fbCamSwitchPulserSearch();
fbCamSwitchPulserSync();
fbInMotionTimer();
fbTestTimer();
fbMotionStage();

IF nTestStep = 78 THEN
    TEST_FINISHED();
ELSIF fbTestTimer.Q THEN
    AssertTrue(FALSE, CONCAT('Timed out at step: ', TO_STRING(nTestStep)));
    TEST_FINISHED();
END_IF
END_METHOD

END_FUNCTION_BLOCK

// ---- POUs/FBs/Common/FB_LimSwStatus.TcPOU
FUNCTION_BLOCK FB_LimSwStatus IMPLEMENTS I_LimSwStatus
VAR_INPUT
END_VAR
VAR_OUTPUT
END_VAR
VAR
    (* Hardware *)
   // NC Forward Limit Switch: TRUE if ok to move
    bLimitForwardEnable AT %I*: BOOL;
    // NC Backward Limit Switch: TRUE if ok to move
    bLimitBackwardEnable AT %I*: BOOL;
    // NO Home Switch: TRUE if at home
    bLimitHome AT %I*: BOOL;
END_VAR

PROPERTY LimitBackwardEnable : BOOL
GET
LimitBackwardEnable := bLimitBackwardEnable;
END_GET
SET
bLimitBackwardEnable := LimitBackwardEnable;
END_SET
END_PROPERTY

PROPERTY LimitForwardEnable : BOOL
GET
LimitForwardEnable := bLimitForwardEnable;
END_GET
SET
bLimitForwardEnable := LimitForwardEnable;
END_SET
END_PROPERTY

PROPERTY LimitHome : BOOL
GET
LimitHome := bLimitHome;
END_GET
SET
bLimitHome := LimitHome;
END_SET
END_PROPERTY

END_FUNCTION_BLOCK

// ---- POUs/FBs/DS402/FB_HomeDS402.TcPOU
FUNCTION_BLOCK FB_HomeDS402 IMPLEMENTS I_HomeDS402
VAR_INPUT
END_VAR
VAR_OUTPUT
END_VAR
VAR
    iMotionLogger : I_MotionLogger;
    //iLimSwStatus : I_LimSwStatus;
    //iHomeShareData : I_HomeShareData ;
    bCommandMoveHome  : BOOL;
    bBusy	: BOOL;
    bDone	: BOOL;
    bError 	: BOOL;
    bAbort   : BOOL;
    bAborted  : BOOL;
    nErrorID : UDINT;
    fOffset  : LREAL;
    fPosition	: LREAL;
    rtDone	: R_TRIG;
    fHomeSpeedFast	: LREAL;
    fHomeSpeedSlow	: LREAL;
    bBit13OpModeSpecific	: BOOL;
    bBit12OpModeSpecific	: BOOL;
    bTargetReached	: BOOL;
    nDriveControl : UINT := 15;
    nModeOfOperation : SINT;
    nModeOfOperationDisplay : SINT;
    nMostRecentModeOfOperation : SINT;
    eHomeMode: E_EpicsHomeCmd :=E_EpicsHomeCmd.AUTOZERO;
    rtExec: R_TRIG;
    ftExec: F_TRIG;
    bMove  : BOOL;
    tonSyncHoming : TON;
    {attribute 'hide'}
    eHomeState	: E_MoveState;
    rtReset: R_TRIG;
    bReset: BOOL;
    sMessage: T_MAXSTRING;
END_VAR

//NB: The calling must pass drive status register.
THIS^.rtExec(CLK:=THIS^.bCommandMoveHome);
THIS^.ftExec(CLK:=THIS^.bCommandMoveHome);
// an interruption can be external i.e, an halt, Reset or a local condition
THIS^.rtReset(CLK:=bReset);
tonSyncHoming(PT:=T#50MS);
CASE THIS^.eHomeMode OF
    E_EpicsHomeCmd.AUTOZERO:
        THIS^.bMove := TRUE;
    E_EpicsHomeCmd.NONE:
        THIS^.bMove := FALSE;
        THIS^.bBusy := THIS^.rtExec.Q;
        THIS^.bDone := NOT THIS^.rtExec.Q;
    ELSE
        THIS^.bMove := FALSE;
END_CASE

IF THIS^.bMove THEN
    IF THIS^.bBusy AND THIS^.ftExec.Q THEN
        THIS^.eHomeState := E_MoveState.ERROR;
        THIS^.bAborted := TRUE;
    END_IF
    CASE eHomeState OF
        // Wait for a rising edge
        E_MoveState.IDLING:
            IF THIS^.rtExec.Q THEN
                THIS^.bDone := FALSE;
                THIS^.bBusy := TRUE;
                THIS^.bError := FALSE;
                THIS^.nErrorID := 0;
                THIS^.bAborted := FALSE;
                THIS^.eHomeState := E_MoveState.INIT;
                // make sure the run flag is clear, this would be the case
                // in EnableMode ->ALWAYS and ModeofOperation ->CSP
                //nDriveControl:=15;
                THIS^.tonSyncHoming.IN := TRUE;
            END_IF
        E_MoveState.INIT:
            // sdo write homing paramters;
            // This mode will be restore after homing
            THIS^.nMostRecentModeOfOperation := nModeOfOperationDisplay;
            nDriveControl:=31;
            // take some time for drive to register above commad and start
            // homming routine.
            IF tonSyncHoming.Q THEN
              eHomeState:=E_MoveState.STARTED;
            END_IF

        E_MoveState.STARTED :
            // this is a comfirmation that routine is ongoing
            IF NOT bTargetReached
               AND NOT bBit13OpModeSpecific THEN
                bBusy:=TRUE;
                bDone:=FALSE;
                eHomeState:=E_MoveState.IN_PROGRESS;
            END_IF
        E_MoveState.IN_PROGRESS :
            // Genral Motion error i.e Following error ?
            IF bBit13OpModeSpecific THEN
                eHomeState:=E_MoveState.ERROR;
            // Reached
            ELSIF bTargetReached
                AND bBit12OpModeSpecific
                AND NOT bBit13OpModeSpecific THEN
                eHomeState:=E_MoveState.REACHED;
            END_IF

        E_MoveState.REACHED:
            bBusy:=FALSE;
            bDone:=TRUE;
            //prepare next move
            nDriveControl:=15;
            // Restore default mode
            //nModeOfOperation:=THIS^.nMostRecentModeOfOperation;
            tonSyncHoming.IN := FALSE;
            eHomeState:=E_MoveState.IDLING;
        E_MoveState.ERROR:
            bError:= TRUE;
            bDone:=FALSE;
            // sdo read in case of error
            bBusy:= FALSE;

    END_CASE
END_IF

IF THIS^.rtReset.Q THEN
    THIS^.bError := FALSE;
    THIS^.nErrorID := 0;
    THIS^.bAborted := FALSE;
    THIS^.sMessage := '';
    THIS^.bReset := FALSE;
    THIS^.eHomeState := E_MoveState.IDLING;
END_IF
//NB: The calling must forward control register for i/o update.
// Reset execute after when done successfull or after abort reset
// this way the done and error condition is latched till next move or global reset.
rtDone(CLK:=bDone);
IF  rtDone.Q  THEN
    THIS^.bCommandMoveHome := FALSE;
END_IF

PROPERTY Aborted : BOOL
GET
Aborted := bAborted;
END_GET
END_PROPERTY

{warning 'Add property implementation'}
PROPERTY Active : BOOL
GET
END_GET
END_PROPERTY

{warning 'add property implementation'}
PROPERTY Busy : BOOL
GET
Busy := THIS^.bBusy;
END_GET
END_PROPERTY

METHOD PUBLIC CallAfterInit
VAR_INPUT
    iMotionLogger : I_MotionLogger;
END_VAR
THIS^.iMotionLogger := iMotionLogger;
END_METHOD

{warning 'Add property implementation'}
PROPERTY CommandMoveHome : BOOL
SET
bCommandMoveHome := CommandMoveHome;
END_SET
END_PROPERTY

{warning 'add property implementation'}
PROPERTY Done : BOOL
GET
Done := THIS^.bDone;
END_GET
END_PROPERTY

PROPERTY DS402Control : UINT
GET
DS402Control := nDriveControl;
END_GET
END_PROPERTY

PROPERTY DS402ModeOfOperation : SINT
GET
DS402ModeOfOperation  := nModeOfOperation;
END_GET
END_PROPERTY

METHOD DS402Status
VAR_INPUT
    ModeOfOperationDisplay : SINT;
    Bit13OpModeSpecific	: BOOL;
    Bit12OpModeSpecific	: BOOL;
    TargetReached	: BOOL;
END_VAR
nModeOfOperationDisplay := ModeOfOperationDisplay;
bBit13OpModeSpecific := Bit13OpModeSpecific;
bBit12OpModeSpecific := Bit12OpModeSpecific;
bTargetReached := TargetReached;
END_METHOD

{warning 'add property implementation'}
PROPERTY Error : BOOL
GET
Error := THIS^.bError;
END_GET
END_PROPERTY

{warning 'add property implementation'}
PROPERTY ErrorID : UDINT
GET
ErrorID := THIS^.nErrorID;
END_GET
END_PROPERTY

//FB_Init is always available implicitly and it is used primarily for initialization.
//The return value is not evaluated. For a specific influence, you can also declare the
//methods explicitly and provide additional code there with the standard initialization
//code. You can evaluate the return value.
METHOD FB_Init: BOOL
VAR_INPUT
    bInitRetains: BOOL; // TRUE: the retain variables are initialized (reset warm / reset cold)
    bInCopyCode: BOOL;  // TRUE: the instance will be copied to the copy code afterward (online change)
    iMotionLogger : I_MotionLogger;
END_VAR
THIS^.iMotionLogger := iMotionLogger;
END_METHOD

{warning 'Add property implementation'}
PROPERTY GlobalReset : BOOL
SET
bReset := GlobalReset;
END_SET
END_PROPERTY

METHOD Home
VAR_INPUT
    Execute	: BOOL;
    HomeSpeedFast	: LREAL;
    HomeSpeedSlow	: LREAL;
END_VAR
THIS^.bCommandMoveHome := Execute;
THIS^.fHomeSpeedFast := HomeSpeedFast;
THIS^.fHomeSpeedSlow := HomeSpeedSlow;
END_METHOD

PROPERTY Message : T_MAXSTRING
GET
Message := sMessage;
END_GET
END_PROPERTY

PROPERTY Mode : E_EpicsHomeCmd
GET
Mode := eHomeMode;
END_GET
SET
eHomeMode := Mode;
END_SET
END_PROPERTY

{warning 'Add property implementation'}
PROPERTY Offset : LREAL
SET
fOffset := Offset;
END_SET
END_PROPERTY

{warning 'Add property implementation'}
PROPERTY Position : LREAL
SET
fPosition := Position;
END_SET
END_PROPERTY

END_FUNCTION_BLOCK

// ---- POUs/FBs/NC/FB_AxisStatusNC.TcPOU
FUNCTION_BLOCK FB_AxisStatusNC IMPLEMENTS I_AxisStatus
VAR_INPUT
END_VAR
VAR_OUTPUT
END_VAR
VAR
    {attribute 'no_copy'}
    AxisRef : REFERENCE TO AXIS_REF;
    bDone : BOOL;
    bBusy    : BOOL;
    sMessage : T_MAXSTRING;
END_VAR

THIS^.AxisRef.ReadStatus();
//THIS^.AxisEnabled();

{warning 'Add property implementation'}
PROPERTY Aborted : BOOL
GET
END_GET
END_PROPERTY

{warning 'Add property implementation'}
PROPERTY Active : BOOL
GET
END_GET
END_PROPERTY

METHOD AxisEnabled : BOOL
// Get a definitive bEnabled reading
CASE THIS^.AxisRef.Status.MotionState OF
    // We are not enabled if there is an issue
    MC_AXISSTATE_UNDEFINED, MC_AXISSTATE_DISABLED, MC_AXISSTATE_ERRORSTOP:
        AxisEnabled := FALSE;
    ELSE
        AxisEnabled := TRUE;
END_CASE
END_METHOD

{warning 'add property implementation'}
PROPERTY AxisID : UDINT
GET
AxisId:=THIS^.AxisRef.NcToPlc.AxisId;
END_GET
END_PROPERTY

{warning 'add property implementation'}
PROPERTY AxisState : Tc2_MC2.MC_AxisStates
GET
AxisState := THIS^.AxisRef.Status.MotionState;
END_GET
END_PROPERTY

{warning 'Add property implementation'}
PROPERTY Busy : BOOL
GET
END_GET
END_PROPERTY

METHOD PUBLIC CallAfterInit
VAR_INPUT
    AxisRef : REFERENCE TO AXIS_REF;
END_VAR
THIS^.AxisRef REF= AxisRef;
END_METHOD

{warning 'Add property implementation'}
PROPERTY Done : BOOL
GET
END_GET
END_PROPERTY

{warning 'add property implementation'}
PROPERTY Error : BOOL
GET
Error := THIS^.AxisRef.Status.Error;
END_GET
END_PROPERTY

{warning 'add property implementation'}
PROPERTY ErrorID : UDINT
GET
ErrorID := THIS^.AxisRef.Status.ErrorID;
END_GET
END_PROPERTY

//FB_Init is always available implicitly and it is used primarily for initialization.
//The return value is not evaluated. For a specific influence, you can also declare the
//methods explicitly and provide additional code there with the standard initialization
//code. You can evaluate the return value.
METHOD FB_Init: BOOL
VAR_INPUT
    bInitRetains: BOOL; // TRUE: the retain variables are initialized (reset warm / reset cold)
    bInCopyCode: BOOL;  // TRUE: the instance will be copied to the copy code afterward (online change)
    AxisRef : REFERENCE TO AXIS_REF;
END_VAR
THIS^.AxisRef REF= AxisRef;
END_METHOD

{warning 'add property implementation'}
PROPERTY InTargetPosition : BOOL
GET
InTargetPosition := THIS^.AxisRef.Status.InTargetPosition;
END_GET
END_PROPERTY

{warning 'add property implementation'}
PROPERTY MeasuredAcceleration : LREAL
GET
MeasuredAcceleration := THIS^.AxisRef.NcToPlc.ActAcc;
END_GET
END_PROPERTY

{warning 'add property implementation'}
PROPERTY MeasuredPosition : LREAL
GET
// (*Actual Position*)
MeasuredPosition:=THIS^.AxisRef.NcToPlc.ActPos;
END_GET
END_PROPERTY

{warning 'add property implementation'}
PROPERTY MeasuredPositionDiff : LREAL
GET
// (*Actual Position Diff*)
MeasuredPositionDiff:=THIS^.AxisRef.NcToPlc.PosDiff;
END_GET
END_PROPERTY

{warning 'add property implementation'}
PROPERTY MeasuredVelocity : LREAL
GET
// (*Actual Velocity*)
MeasuredVelocity:=THIS^.AxisRef.NcToPlc.ActVelo;
END_GET
END_PROPERTY

PROPERTY Message : T_MAXSTRING
GET
Message := sMessage;
END_GET
END_PROPERTY

{warning 'add property implementation'}
PROPERTY NegativeMotionIsEnabled : BOOL
GET
NegativeMotionIsEnabled := THIS^.AxisRef.Status.NegativeDirection;
END_GET
END_PROPERTY

{warning 'add property implementation'}
PROPERTY PositiveMotionIsEnabled : BOOL
GET
PositiveMotionIsEnabled := THIS^.AxisRef.Status.PositiveDirection;
END_GET
END_PROPERTY

PROPERTY StandStill : BOOL
GET
StandStill := THIS^.AxisRef.Status.StandStill;
END_GET
END_PROPERTY

{warning 'Add property implementation'}
PROPERTY Stopped : BOOL
GET
Stopped := THIS^.AxisRef.Status.HasBeenStopped;
END_GET
END_PROPERTY

END_FUNCTION_BLOCK

// ---- POUs/FBs/NC/FB_BrakeNC.TcPOU
FUNCTION_BLOCK FB_BrakeNC IMPLEMENTS I_Brake
VAR
    // Determines when we automatically disengage the brake
    eBrakeMode: E_StageBrakeMode:=E_StageBrakeMode.IF_ENABLED;
    // NC Brake Output: TRUE to release brake
    bBrakeRelease AT %Q*: BOOL;
    // pass it an AXIS_REF.
    eAxisState : MC_AxisStates;

END_VAR

// Handle the brake. TRUE means brake disabled/released
IF eBrakeMode <> E_StageBrakeMode.NO_BRAKE THEN
    CASE eAxisState OF
        MC_AXISSTATE_UNDEFINED,
        MC_AXISSTATE_DISABLED,
        MC_AXISSTATE_ERRORSTOP:
            bBrakeRelease := FALSE;
        MC_AXISSTATE_STANDSTILL:
            IF eBrakeMode = E_StageBrakeMode.IF_MOVING THEN
                bBrakeRelease := FALSE;
            ELSE
                bBrakeRelease := TRUE;
            END_IF
        ELSE
            bBrakeRelease := TRUE;
    END_CASE
ELSE
    bBrakeRelease := TRUE;
END_IF

{warning 'add property implementation'}
PROPERTY Aborted : BOOL
GET
END_GET
END_PROPERTY

{warning 'Add property implementation'}
PROPERTY Active : BOOL
GET
END_GET
END_PROPERTY

PROPERTY AxisState : MC_AxisStates
SET
eAxisState := AxisState;
END_SET
END_PROPERTY

PROPERTY BrakeMode : E_StageBrakeMode
GET
END_GET
SET
eBrakeMode := BrakeMode;
END_SET
END_PROPERTY

PROPERTY BrakeRelease : BOOL
GET
BrakeRelease := bBrakeRelease;
END_GET
END_PROPERTY

{warning 'add property implementation'}
PROPERTY Busy : BOOL
GET
END_GET
END_PROPERTY

{warning 'add property implementation'}
PROPERTY Done : BOOL
GET
END_GET
END_PROPERTY

{warning 'Add property implementation'}
PROPERTY Error : BOOL
GET
END_GET
END_PROPERTY

{warning 'Add property implementation'}
PROPERTY ErrorID : UDINT
GET
END_GET
END_PROPERTY

{warning 'Add property implementation'}
PROPERTY Message : T_MAXSTRING
GET
END_GET
END_PROPERTY

END_FUNCTION_BLOCK

// ---- POUs/FBs/NC/FB_ParamsSaveRestoreNC.TcPOU
{attribute 'call_after_init'}
FUNCTION_BLOCK FB_ParamsSaveRestoreNC IMPLEMENTS I_ParamSaveRestore
VAR_INPUT
END_VAR
VAR_OUTPUT
END_VAR
VAR
    {attribute 'no_copy'}
    AxisRef : REFERENCE TO AXIS_REF;
    iPersistentDataStorage : I_PersistentDataStorage;

    // save and restore
    fbSetPos: MC_SetPosition;
    bClearPositionLag : BOOL := TRUE;

    nLatchErrId : BOOL;
    bRestoreDone 	: BOOL;
    bRestoreError 	: BOOL;
    nRestoreErrorID : UDINT;
    // save and Restore
    RestoreTimer: TON;
    bRestoreInit: BOOL;
    bRestoreLoad: BOOL;
    nLatchError: UDINT;
    bEncError: BOOL;
    tRetryDelay: TIME := T#1S;
    tRefreshDelay: TIME := T#1S;
    bUpdateEnable : BOOL;
    bExecute : BOOL;
    nMaxRetries: UINT := 10;
    nCurrTries: UINT := 0;
    bRestoreWaitRetry: BOOL;
    tonRestoreRetry: TON;
    tRefreshTime : TIME := T#1S;
    bError				: BOOL;
    nErrorId			: UDINT:=0;
    sMessage : T_MAXSTRING;

    bSaveEnabled	: BOOL := TRUE;
    bDone : BOOL;
    bBusy    : BOOL;
END_VAR

VAR PERSISTENT
    {attribute 'conditionalshow'}
    bSaved: BOOL;
    {attribute 'conditionalshow'}
    fSavedPosition: LREAL;
END_VAR

IF NOT __ISVALIDREF(THIS^.AxisRef) THEN
    RETURN;
END_IF

THIS^.AxisRef.ReadStatus();

// Save Encoder position
// needs some pre-conditions to use persistent storage
IF bSaveEnabled THEN
    // Check ST_MotionStage for an encoder error (range 0x44nn)
    bEncError:= AxisRef.Status.Error AND  ( AxisRef.Status.ErrorID  >= 16#4400  AND AxisRef.Status.ErrorID <= 16#44FF );
    // Do not save if we're currently loading or if there is an encoder error
    IF NOT bRestoreLoad AND NOT bEncError AND NOT bRestoreWaitRetry THEN
        fSavedPosition := AxisRef.NcToPlc.ActPos;
        // This persistent variable lets us check if anything was saved
        // It will be TRUE at startup if we have saved values
        bSaved := TRUE;
        (*
            use this with a timer of a change threshold on the fActPosition
            to trigger a save from this PLC program. otherwise this will be a spamming
            persistence, filling up the disk.
        *)
        //iPersistentDataStorage.TriggerWriteOfPersistentData := bSaveEnabled;
    END_IF
END_IF

{warning 'Add property implementation'}
PROPERTY Aborted : BOOL
GET
END_GET
END_PROPERTY

{warning 'Add property implementation'}
PROPERTY Active : BOOL
GET
END_GET
END_PROPERTY

{warning 'Add property implementation'}
PROPERTY Busy : BOOL
GET
END_GET
END_PROPERTY

METHOD PUBLIC CallAfterInit
VAR_INPUT
    AxisRef : REFERENCE TO AXIS_REF;
    iPersistentDataStorage : I_PersistentDataStorage;
END_VAR
THIS^.AxisRef REF= AxisRef;
THIS^.iPersistentDataStorage := iPersistentDataStorage;
END_METHOD

{warning 'Add property implementation'}
PROPERTY Done : BOOL
GET
END_GET
END_PROPERTY

{warning 'add property implementation'}
PROPERTY Error : BOOL
GET
Error := bError;
END_GET
END_PROPERTY

{warning 'add property implementation'}
PROPERTY ErrorID : UDINT
GET
ErrorID := nErrorID;
END_GET
END_PROPERTY

//FB_Init is always available implicitly and it is used primarily for initialization.
//The return value is not evaluated. For a specific influence, you can also declare the
//methods explicitly and provide additional code there with the standard initialization
//code. You can evaluate the return value.
METHOD FB_Init: BOOL
VAR_INPUT
    bInitRetains: BOOL; // TRUE: the retain variables are initialized (reset warm / reset cold)
    bInCopyCode: BOOL;  // TRUE: the instance will be copied to the copy code afterward (online change)
    AxisRef : REFERENCE TO AXIS_REF;
    iPersistentDataStorage : I_PersistentDataStorage;
END_VAR
THIS^.AxisRef REF= AxisRef;
THIS^.iPersistentDataStorage := iPersistentDataStorage;
END_METHOD

PROPERTY Message : T_MAXSTRING
GET
Message := sMessage;
END_GET
END_PROPERTY

{attribute 'call_after_init'}
METHOD RestoreAxisParams
// Trigger a load if anything was saved at all
IF NOT bRestoreInit THEN
    bRestoreInit := TRUE;
    bRestoreLoad S= bSaved;
    fbSetPos.Options.ClearPositionLag := TRUE;
END_IF

// Set our position if bRestoreLoad is true
fbSetPos( Axis:=THIS^.AxisRef, Execute:=bRestoreLoad, Position:=fSavedPosition);

// Only load once, at startup
bRestoreLoad R= fbSetPos.Done OR fbSetPos.Error;

IF fbSetPos.Error THEN
    // Keep the error latched, it can disappear if Execute is set to FALSE
    nLatchError := fbSetPos.ErrorID;
    nCurrTries := nCurrTries + 1;
    IF nCurrTries >= nMaxRetries THEN
    // Alert the user that something has gone wrong
    bError := TRUE;
        nErrorId := nLatchError;
        sMessage := 'Error loading previously saved position.';
    ELSE
        // Reset the FB for the next retry
        fbSetPos( Axis:=THIS^.AxisRef, Execute:=bRestoreLoad, Position:=fSavedPosition);
        // Try again
        bRestoreWaitRetry := TRUE;
    END_IF
ELSE
    THIS^.bRestoreDone := TRUE;
END_IF

tonRestoreRetry( IN := bRestoreWaitRetry, PT := tRetryDelay);
bRestoreLoad S= tonRestoreRetry.Q;
bRestoreWaitRetry R= tonRestoreRetry.Q;
END_METHOD

{warning 'add property implementation'}
PROPERTY RestoreDone : BOOL
GET
END_GET
END_PROPERTY

METHOD SaveAxisParams
VAR_INPUT
    Enable	: BOOL;
END_VAR
THIS^.bSaveEnabled := Enable;
END_METHOD

{warning 'add property implementation'}
PROPERTY SavedPosition : LREAL
GET
SavedPosition := fSavedPosition;
END_GET
END_PROPERTY

END_FUNCTION_BLOCK

// ---- POUs/FBs/NC/FB_ReadParameterNC.TcPOU
(*
    Read and refresh axis parameters
*)
FUNCTION_BLOCK FB_ReadParameterNC IMPLEMENTS I_ReadParameter
VAR
    {attribute 'no_copy'}
    AxisRef : REFERENCE TO AXIS_REF;
	iMotionLogger : I_MotionLogger := 0;
    // NC parameters that are exposed with pytmc pragmas
    {attribute 'pytmc' := '
        pv: PLC:AxisPar
        io: i
        field: DESC Axis configuration parameters in the numerical controller.
    '}
    stAxisParametersExposed : ST_AxisParameterSetExposed;
    // MC_ReadParameterSet Output
    fbMcReadParams: MC_ReadParameterSet;
    {attribute 'hide'}
    stAxisParameters: ST_AxisParameterSet;
    {attribute 'hide'}
    NCParamsTimer : TON;
    {attribute 'hide'}
    bExecParamsRead: BOOL;
    {attribute 'hide'}
    bAxisParamsInit: BOOL;
    {attribute 'hide'}
	bEnable : BOOL;
    {attribute 'hide'}
	rtError: R_TRIG;
END_VAR

// Periodic update of NC parameters
NCParamsTimer( IN:=NOT bExecParamsRead, PT:=T#1S);

bExecParamsRead S= NCParamsTimer.Q;

fbMcReadParams(
    Parameter:=stAxisParameters,
    Axis:=AxisRef );
	
// Copy axis parameters that we want to expose to the EPICS layer.
stAxisParametersExposed.bCtrlEnablePosDiffControl     := stAxisParameters.bCtrlEnablePosDiffControl;
stAxisParametersExposed.bEncEnableSoftEndMaxControl   := stAxisParameters.bEncEnableSoftEndMaxControl;
stAxisParametersExposed.bEncEnableSoftEndMinControl   := stAxisParameters.bEncEnableSoftEndMinControl;
stAxisParametersExposed.fAccelerationMax              := stAxisParameters.fAccelerationMax;
stAxisParametersExposed.fCtrlPosDiffMax               := stAxisParameters.fCtrlPosDiffMax;
stAxisParametersExposed.fCtrlPosDiffMaxTime           := stAxisParameters.fCtrlPosDiffMaxTime;
stAxisParametersExposed.fDecelerationMax              := stAxisParameters.fDecelerationMax;
stAxisParametersExposed.fEncSoftEndMax                := stAxisParameters.fEncSoftEndMax;
stAxisParametersExposed.fEncSoftEndMin                := stAxisParameters.fEncSoftEndMin;
stAxisParametersExposed.fVeloMaximum                  := stAxisParameters.fVeloMaximum;
stAxisParametersExposed.fEncOffset               	  := stAxisParameters.fEncOffset;
stAxisParametersExposed.fEncScaleFactorInternal       := stAxisParameters.fEncScaleFactorInternal;

bExecParamsRead R= fbMcReadParams.Done OR fbMcReadParams.Error;
bAxisParamsInit S= fbMcReadParams.Done;

rtError(CLK:=fbMcReadParams.Error);
IF rtError.Q THEN
	iMotionLogger.Logger(Message := iMotionLogger.ErrorCodeLookup(fbMcReadParams.ErrorID), Level := E_MotionLogLevel.ERROR, Source := 'ReadParams');	
END_IF

PROPERTY AxisReadParamsInit : BOOL
GET
AxisReadParamsInit := bAxisParamsInit;
END_GET
END_PROPERTY

PROPERTY Busy : BOOL
GET
Busy := fbMcReadParams.Busy;
END_GET
END_PROPERTY

METHOD PUBLIC CallAfterInit
VAR_INPUT
    AxisRef : REFERENCE TO AXIS_REF;
	iMotionLogger : I_MotionLogger;
END_VAR
THIS^.AxisRef REF= AxisRef;
THIS^.iMotionLogger := iMotionLogger;
END_METHOD

PROPERTY Done : BOOL
GET
Done := fbMcReadParams.Done;
END_GET
END_PROPERTY

PROPERTY Error : BOOL
GET
Error := fbMcReadParams.Error;
END_GET
END_PROPERTY

PROPERTY ErrorID : UDINT
GET
ErrorID := fbMcReadParams.ErrorID;
END_GET
END_PROPERTY

//FB_Init is always available implicitly and it is used primarily for initialization.
//The return value is not evaluated. For a specific influence, you can also declare the
//methods explicitly and provide additional code there with the standard initialization
//code. You can evaluate the return value.
METHOD FB_Init: BOOL
VAR_INPUT
    bInitRetains: BOOL; // TRUE: the retain variables are initialized (reset warm / reset cold)
    bInCopyCode: BOOL;  // TRUE: the instance will be copied to the copy code afterward (online change)
    AxisRef : REFERENCE TO AXIS_REF;
	iMotionLogger : I_MotionLogger := 0;	
END_VAR
THIS^.AxisRef REF= AxisRef;
THIS^.iMotionLogger := iMotionLogger;
END_METHOD

PROPERTY Message : T_MAXSTRING
GET
END_GET
END_PROPERTY

METHOD ReadParameters
VAR_INPUT
    Enable : BOOL;
    RefreshDelay : TIME;
END_VAR
fbMcReadParams(
    Parameter:=THIS^.stAxisParameters,
    Axis:=THIS^.AxisRef,
    Execute:= Enable AND THIS^.bExecParamsRead );

NCParamsTimer.PT:=RefreshDelay;
END_METHOD

END_FUNCTION_BLOCK

// ---- POUs/FBs/NC/FB_WriteParameterNC.TcPOU
FUNCTION_BLOCK FB_WriteParameterNC IMPLEMENTS I_WriteParameter
VAR
    {attribute 'no_copy'}
    AxisRef : REFERENCE TO AXIS_REF;
    fbMcWriteParameter : MC_WriteParameter;
    bExecute : BOOL;
    bError	: BOOL;
    nErrorId : UDINT:=0;
    sMessage : T_MAXSTRING;
    bDone : BOOL;
    bBusy    : BOOL;
    nParameterNumber : MC_AxisParameter;
    fParameterValue	: LREAL;
    rtDone : R_TRIG;
END_VAR

IF NOT __ISVALIDREF(THIS^.AxisRef) THEN
    RETURN;
END_IF

THIS^.AxisRef.ReadStatus();

(*Do not change a moving axis parameter*)
fbMcWriteParameter(	Axis:=THIS^.AxisRef,
                    Execute:=(THIS^.bExecute AND THIS^.AxisRef.Status.NotMoving),
                    ParameterNumber:=THIS^.nParameterNumber,
                    Value:=THIS^.fParameterValue,
                    Done=>THIS^.bDone,
                    Busy=>THIS^.bBusy,
                    Error=>THIS^.bError,
                    ErrorID=>THIS^.nErrorID
                  );

// Reset execute after when done successfull or after abort reset
// this way the done and error condition is latched till next move or global reset.
rtDone(CLK:=bDone);
IF  rtDone.Q THEN
    THIS^.bExecute := FALSE;
END_IF

{warning 'Add property implementation'}
PROPERTY Aborted : BOOL
GET
END_GET
END_PROPERTY

{warning 'Add property implementation'}
PROPERTY Active : BOOL
GET
END_GET
END_PROPERTY

{warning 'Add property implementation'}
PROPERTY Busy : BOOL
GET
Busy := bBusy;
END_GET
END_PROPERTY

METHOD PUBLIC CallAfterInit
VAR_INPUT
    AxisRef : REFERENCE TO AXIS_REF;
END_VAR
THIS^.AxisRef REF= AxisRef;
END_METHOD

{warning 'Add property implementation'}
PROPERTY Done : BOOL
GET
Done := bDone;
END_GET
END_PROPERTY

{warning 'add property implementation'}
PROPERTY Error : BOOL
GET
Error := bError;
END_GET
END_PROPERTY

{warning 'add property implementation'}
PROPERTY ErrorID : UDINT
GET
ErrorID := nErrorID;
END_GET
END_PROPERTY

//FB_Init is always available implicitly and it is used primarily for initialization.
//The return value is not evaluated. For a specific influence, you can also declare the
//methods explicitly and provide additional code there with the standard initialization
//code. You can evaluate the return value.
METHOD FB_Init: BOOL
VAR_INPUT
    bInitRetains: BOOL; // TRUE: the retain variables are initialized (reset warm / reset cold)
    bInCopyCode: BOOL;  // TRUE: the instance will be copied to the copy code afterward (online change)
    AxisRef : REFERENCE TO AXIS_REF;
END_VAR
THIS^.AxisRef REF= AxisRef;
END_METHOD

PROPERTY Message : T_MAXSTRING
GET
Message := sMessage;
END_GET
END_PROPERTY

METHOD WriteParameter
VAR_INPUT
    Execute         : BOOL;
    ParameterNumber : MC_AxisParameter;
    ParameterValue	: LREAL;
END_VAR
THIS^.bExecute := Execute;
THIS^.nParameterNumber := ParameterNumber;
THIS^.fParameterValue	:= ParameterValue;
END_METHOD

END_FUNCTION_BLOCK

// ---- Test/HARD_TEST.TcPOU
PROGRAM HARD_TEST
VAR
    fbAxisRef : AXIS_REF;
	fbPersistentDataStorage :  FB_PersistentDataStorage;
   	fbMotionStage : FB_MotionStageNC(	sName := 'Test2',
                                        AxisRef := fbAxisRef,
                                        iPersistentDataStorage := fbPersistentDataStorage
                                    ) ;
    nTestStep : INT;
END_VAR


// fbPower.Power(	
// 	Enable:=TRUE,
// 	Enable_Positive:=TRUE,
// 	Enable_Negative:=TRUE,
// 	Override:=100.0
// );

				  
CASE nTestStep OF
    0:
//        fbMoveAbsolute.MoveAbsolute(
//             Position := 10000.0,
//             Velocity := 50.0,
//             Acceleration := 500.0,
//             Deceleration := 500.0
//         );
//         fbMotionStage.AbsoluteMove(
//             Position := 1000.0,
//             Velocity := 50.0,
//             Acceleration := 200.0,
//             Deceleration := 200.0
//         );
 		nTestStep := nTestStep + 1;

END_CASE
fbMotionStage();
//fbReset();
//fbMoveAbsolute();

END_PROGRAM

// ---- Test/CONTAINER_TEST.TcPOU
PROGRAM CONTAINER_TEST
VAR
    fbAxisRef : AXIS_REF;
	fbMotionLogger : FB_MotionLogger_TestDouble;
	fbPower: FB_PowerNC(AxisRef:=fbAxisRef, iMotionLogger:=fbMotionLogger);
	fbMcReset 	: MC_Reset;
	fbMcPower : MC_Power;
    fbMcHome : MC_Home;
    fbMcSetPosition : MC_SetPosition;
	bLimPositive : BOOL := TRUE;
	bLimNegative : BOOL := TRUE;
	bTriggerHome : BOOL;
	bHomingOverride: BOOL := TRUE;
    nTestStep : INT;
	bEnable: BOOL;
	bReset: BOOL;
END_VAR




fbMcHome.bCalibrationCam := NOT bLimNegative;
				  
CASE nTestStep OF
    0:
        fbMcHome.HomingMode := MC_HomingMode.MC_DefaultHoming;
        fbMcHome.Options.SearchDirection := MC_Direction.MC_Negative_Direction;
        fbMcHome.Options.SyncDirection := MC_Direction.MC_Positive_Direction;
        fbMcHome.Options.ClearPositionLag := TRUE;
		nTestStep := 1;
	1:
		IF fbMcPower.Status THEN
			fbMcHome.Execute := TRUE;
			nTestStep := 2;			
		END_IF


END_CASE
fbMcReset(   Axis := fbAxisRef,
             Execute := bReset );

fbMcPower(
    Axis :=  fbAxisRef,
    Enable := bEnable,
    Enable_Positive := bHomingOverride OR bLimPositive,
    Enable_Negative := bHomingOverride OR bLimNegative,
    Override :=100.0
);
fbMcHome( Axis := fbAxisRef, Position := 5.0  );

END_PROGRAM

// ---- Test/TestDouble/FB_EpicsMotionParamsStatus_TestDouble.TcPOU
FUNCTION_BLOCK FB_EpicsMotionParamsStatus_TestDouble IMPLEMENTS I_EpicsMotionParamsStatus
VAR
END_VAR

{warning 'Add method implementation '}
METHOD MotionParamsAndStatus
VAR_INPUT
	PowerEnabled	: BOOL;
	PowerIsEnabled	: BOOL;
	Execute	: BOOL;
	LimHome	: BOOL;
	MoveBackwardEnabled	: BOOL;
	MoveForwardEnabled	: BOOL;
	MeasuredPositionDiff	: LREAL;
	MeasuredPosition	: LREAL;
	MeasuredVelocity	: LREAL;
	PowerOverride	: LREAL;
	Busy	: BOOL;
	HomeDone	: BOOL;
	MotionAxisId : UDINT;
END_VAR
END_METHOD

END_FUNCTION_BLOCK
